RoboDK station: Kuka_KR3_R540.rdk

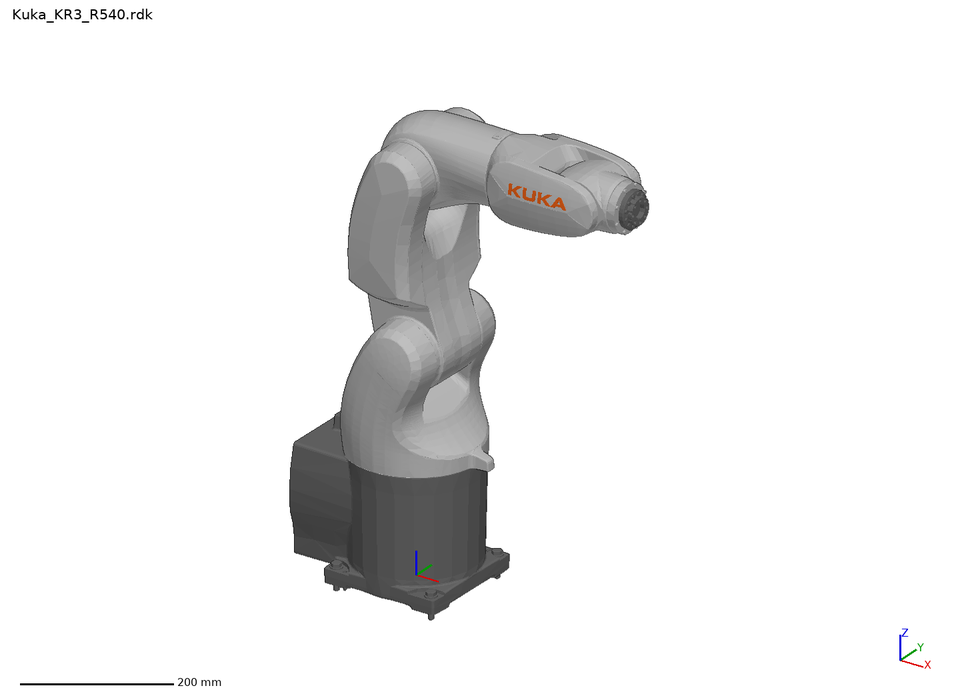
[picture v0: the station drawn from its stored meshes, robots at their saved joint values, targets as dots, program paths as lines]
Station Kuka_KR3 R540 (saved by RoboDK 5.6.4). Poses are relative to the parent item; angles as X-Y-Z fixed-axis rotations.
  - frame KUKA KR 3 R540 Base at (0, 0, 0) mm
    - robot KUKA KR 3 R540: 6 axes, payload 3 kg, reach 541 mm, repeatability 0.02 mm, weight 26 kg
        modified DH rows (alpha deg, a mm, theta deg, d mm): 0, 0, 0, 345; -90, 20, 0, 0; 0, 260, -90, 0; -90, 20, 0, 260; 90, 0, 0, 0; -90, 0, 180, 75
        joint limits [-170, -170, -110, -175, -120, -350] to [170, 50, 155, 175, 120, 350]; home [0, -90, 90, 0, 0, 0]; saved at [0, -90, 90, 0.56, 0, -0.56]
